# EPICS autosave request: iocBoot/iocrsfsl/auto_settings_rsfsl.req
file "rsfsl_settings.req",                P=$(P),  R=$(R)
